(* CoDeSys 2.3.9.41 project: Armen_1.pro *)
(* Libraries: Util.lib 18.5.10 15:14:28, STANDARD.LIB 4.10.05 11:14:46, IECSFC.LIB 13.4.06 15:51:28, SYSLIBTIME.LIB 20.2.06 12:31:16, SYSTASKINFO.LIB 20.2.06 12:31:38, ANALYZATION.LIB 5.10.99 09:05:06, SYSLIBCALLBACK.LIB 20.2.06 12:31:08, PID_Regulators.lib 28.12.06 16:47:54 *)

(* PLC configuration (modules and I/O channels)
Fast discrete inputs [I_SIMPLE_INPUT] node 0, in %IB0 out %QB0 {ChannellName = Fast discrete inputs; Filtrationtime = 10000}
  AT %IX0.0 [BitInput] Discrete input 1 {ChannellName = Enter name}
  AT %IX0.1 [BitInput] Discrete input 2 {ChannellName = Enter name}
AT %IB1.0 [ByteInput] 8 discrete inputs {ChannellName = Enter name}
AT %IB1.1 [ByteInput] 8 discrete inputs {ChannellName = Enter name}
Fan AT %QX2.0 [BitOutput] Fast discrete output 1 {ChannellName = Enter name}
Hot_fan AT %QX2.1 [BitOutput] Fast discrete output 2 {ChannellName = Enter name}
Fan_wall AT %QX2.2 [BitOutput] Fast discrete output 3 {ChannellName = Enter name}
Light_out AT %QX2.3 [BitOutput] Fast discrete output 4 {ChannellName = Enter name}
AT %QB3.0 [ByteOutput] 8 discrete outputs {ChannellName = Enter name}
AT %IX4.0 [BitInput] Special input {ChannellName = Enter name}
AT %QX5.0 [BitOutput] Special output {ChannellName = Enter name}
RS-232 [COM2_USART] node 0, in %IB6.0.0 out %QB6.0.0 {ChannellName = RS-232; CommunicationSpeed = 57600; Parity = NO PARITY CHECK; BitLength = 8 bits; StopLength = One stop bit; InterfaceType = RS232; FrameOriented = RTU; Timeout = 0; Visibility = No}
AT %QB6.1.0 [ByteOutput] {ChannellName = Enter name}
AT %QB6.2.0 [ByteOutput] {ChannellName = Enter name}
AT %QB6.3.0 [ByteOutput] {ChannellName = Enter name}
8 bits [8Bit] node 4, in %IB6.4 out %QB6.4 {ChannellName = 8 bit}
  AT %QB6.4.0 [ByteOutput] {ChannellName = Enter name}
8 bits [8Bit] node 5, in %IB6.5 out %QB6.5 {ChannellName = 8 bit}
  AT %QB6.5.0 [ByteOutput] {ChannellName = Enter name}
8 bits [8Bit] node 6, in %IB6.6 out %QB6.6 {ChannellName = 8 bit}
  AT %QB6.6.0 [ByteOutput] {ChannellName = Enter name}
2 byte [Register] node 7, in %IB6.7 out %QB6.7 {ChannellName = 2 byte}
  Hour_p AT %QW6.7.0 [WordOutput] {ChannellName = Enter name}
2 byte [Register] node 8, in %IB6.8 out %QB6.8 {ChannellName = 2 byte}
  Min_p AT %QW6.8.0 [WordOutput] {ChannellName = Enter name}
2 byte [Register] node 9, in %IB6.9 out %QB6.9 {ChannellName = 2 byte}
  FanWall_t_start AT %QW6.9.0 [WordOutput] {ChannellName = Enter name}
2 byte [Register] node 10, in %IB6.10 out %QB6.10 {ChannellName = 2 byte}
  FanWall_t_stop AT %QW6.10.0 [WordOutput] {ChannellName = Enter name}
2 byte [Register] node 11, in %IB6.11 out %QB6.11 {ChannellName = 2 byte}
  Wind_set AT %QW6.11.0 [WordOutput] {ChannellName = Enter name}
2 byte [Register] node 12, in %IB6.12 out %QB6.12 {ChannellName = 2 byte}
  Wind_Hyst AT %QW6.12.0 [WordOutput] {ChannellName = Enter name}
2 byte [Register] node 13, in %IB6.13 out %QB6.13 {ChannellName = 2 byte}
  Fan_set AT %QW6.13.0 [WordOutput] {ChannellName = Enter name}
2 byte [Register] node 14, in %IB6.14 out %QB6.14 {ChannellName = 2 byte}
  Fan_Hyst AT %QW6.14.0 [WordOutput] {ChannellName = Enter name}
2 byte [Register] node 15, in %IB6.15 out %QB6.15 {ChannellName = 2 byte}
  Hot_set AT %QW6.15.0 [WordOutput] {ChannellName = Enter name}
2 byte [Register] node 16, in %IB6.16 out %QB6.16 {ChannellName = 2 byte}
  Hot_Hyst AT %QW6.16.0 [WordOutput] {ChannellName = Enter name}
2 byte [Register] node 17, in %IB6.17 out %QB6.17 {ChannellName = 2 byte}
  Cold_set AT %QW6.17.0 [WordOutput] {ChannellName = Enter name}
2 byte [Register] node 18, in %IB6.18 out %QB6.18 {ChannellName = 2 byte}
  Cold_hyst AT %QW6.18.0 [WordOutput] {ChannellName = Enter name}
2 byte [Register] node 19, in %IB6.19 out %QB6.19 {ChannellName = 2 byte}
  m_Light_on AT %QW6.19.0 [WordOutput] {ChannellName = Enter name}
2 byte [Register] node 20, in %IB6.20 out %QB6.20 {ChannellName = 2 byte}
  h_light_on AT %QW6.20.0 [WordOutput] {ChannellName = Enter name}
2 byte [Register] node 21, in %IB6.21 out %QB6.21 {ChannellName = 2 byte}
  m_light_off AT %QW6.21.0 [WordOutput] {ChannellName = Enter name}
2 byte [Register] node 22, in %IB6.22 out %QB6.22 {ChannellName = 2 byte}
  h_light_off AT %QW6.22.0 [WordOutput] {ChannellName = Enter name}
2 byte [Register] node 23, in %IB6.23 out %QB6.23 {ChannellName = 2 byte}
  t_tep_i AT %QW6.23.0 [WordOutput] {ChannellName = Enter name}
2 byte [Register] node 24, in %IB6.24 out %QB6.24 {ChannellName = 2 byte}
  v_tep_i AT %QW6.24.0 [WordOutput] {ChannellName = Enter name}
2 byte [Register] node 25, in %IB6.25 out %QB6.25 {ChannellName = 2 byte}
  t_ul_i AT %QW6.25.0 [WordOutput] {ChannellName = Enter name}
2 byte [Register] node 26, in %IB6.26 out %QB6.26 {ChannellName = 2 byte}
  v_ul_i AT %QW6.26.0 [WordOutput] {ChannellName = Enter name}
2 byte [Register] node 27, in %IB6.27 out %QB6.27 {ChannellName = 2 byte}
  AT %QW6.27.0 [WordOutput] {ChannellName = Enter name}
2 byte [Register] node 28, in %IB6.28 out %QB6.28 {ChannellName = 2 byte}
  AT %QW6.28.0 [WordOutput] {ChannellName = Enter name}
2 byte [Register] node 29, in %IB6.29 out %QB6.29 {ChannellName = 2 byte}
  AT %QW6.29.0 [WordOutput] {ChannellName = Enter name}
2 byte [Register] node 30, in %IB6.30 out %QB6.30 {ChannellName = 2 byte}
  AT %QW6.30.0 [WordOutput] {ChannellName = Enter name}
2 byte [Register] node 31, in %IB6.31 out %QB6.31 {ChannellName = 2 byte}
  AT %QW6.31.0 [WordOutput] {ChannellName = Enter name}
4 byte [FourBytes] node 32, in %IB6.32 out %QB6.32 {ChannellName = 4 byte}
  AT %QD6.32.0 [DWordOutput] {ChannellName = Enter name}
AT %QD7.0 [DWordOutput] Last address {ChannellName = Enter name}
AT %QW7.1 [WordOutput] Last error {ChannellName = Enter name}
RS-485-1 [COM1_USART] node 0, in %IB7.0 out %QB7.0 {ChannellName = RS-485-1; CommunicationSpeed = 38400; Parity = NO PARITY CHECK; BitLength = 8 bits; StopLength = One stop bit; InterfaceType = RS485; FrameOriented = ASCII; Timeout = 0; Visibility = No}
Universal Modbus device [ID2000] node 1, in %IB7.1 out %QB7.1 {ChannellName = Universal Modbus device; ModuleIP = 10:0:0:223; ServiceTimeout = 150; TCPport = 502; NetMode = Serial; ModuleSlaveAddress = 2; RequestType = By poll time; PeriodOfService = 100; Visibility = No; RepeatCounter = 0; ByteSequence = Trace_mode}
  AT %QB7.1.0 [ComChannel] Command (0xff - Start) {ChannellName = Enter name}
Wind AT %QD7.1.0.0 [FloatOutput] {ChannellName = Enter name}
AT %QD7.1.1.0 [FloatOutput] {ChannellName = Enter name}
Universal Modbus device [ID2000] node 2, in %IB7.2 out %QB7.2 {ChannellName = Universal Modbus device; ModuleIP = 10:0:0:223; ServiceTimeout = 150; TCPport = 502; NetMode = Serial; ModuleSlaveAddress = 1; RequestType = By poll time; PeriodOfService = 100; Visibility = No; RepeatCounter = 0; ByteSequence = Trace_mode}
  AT %QB7.2.0 [ComChannel] Command (0xff - Start) {ChannellName = Enter name}
t_tep AT %QW7.2.0.0 [WordOutput] {ChannellName = Enter name}
v_tep AT %QW7.2.1.0 [WordOutput] {ChannellName = Enter name}
Universal Modbus device [ID2000] node 3, in %IB7.3 out %QB7.3 {ChannellName = Universal Modbus device; ModuleIP = 10:0:0:223; ServiceTimeout = 150; TCPport = 502; NetMode = Serial; ModuleSlaveAddress = 1; RequestType = By poll time; PeriodOfService = 100; Visibility = No; RepeatCounter = 0; ByteSequence = Trace_mode}
  AT %QB7.3.0 [ComChannel] Command (0xff - Start) {ChannellName = Enter name}
t_ul AT %QW7.3.0.0 [WordOutput] {ChannellName = Enter name}
v_ul AT %QW7.3.1.0 [WordOutput] {ChannellName = Enter name}
AT %QB7.4.0 [ComChannel] Command (0xff - Start) {ChannellName = Enter name}
PR100_in AT %QW7.4.0.0 [WordOutput] {ChannellName = Enter name}
PR100_out AT %QW7.4.1.0 [WordOutput] {ChannellName = Enter name}
Real input module [ID2007] node 2, in %IB7.4.2 out %QB7.4.2 {ChannellName = float input module; ModbusAddress = 0; Command_read_regs = Read holding Registers  (0x03); Visibility = No}
  AT %QD7.4.2.0 [FloatOutput] {ChannellName = Enter name}
Real input module [ID2007] node 3, in %IB7.4.3 out %QB7.4.3 {ChannellName = float input module; ModbusAddress = 0; Command_read_regs = Read holding Registers  (0x03); Visibility = No}
  AT %QD7.4.3.0 [FloatOutput] {ChannellName = Enter name}
*)

(* POU PLC_PRG, CFC *)
PROGRAM PLC_PRG
VAR
	Tof_Cold: TOF;
	FanWall: BLINK;
	Window_contr: HYSTERESIS;
	Hot_contr: HYSTERESIS;
	Cold_contr: HYSTERESIS;
	Tof_hot: TOF;

	Tof_wind: TOF;
	Window2_tim,Window2_tim_2: TON;
END_VAR
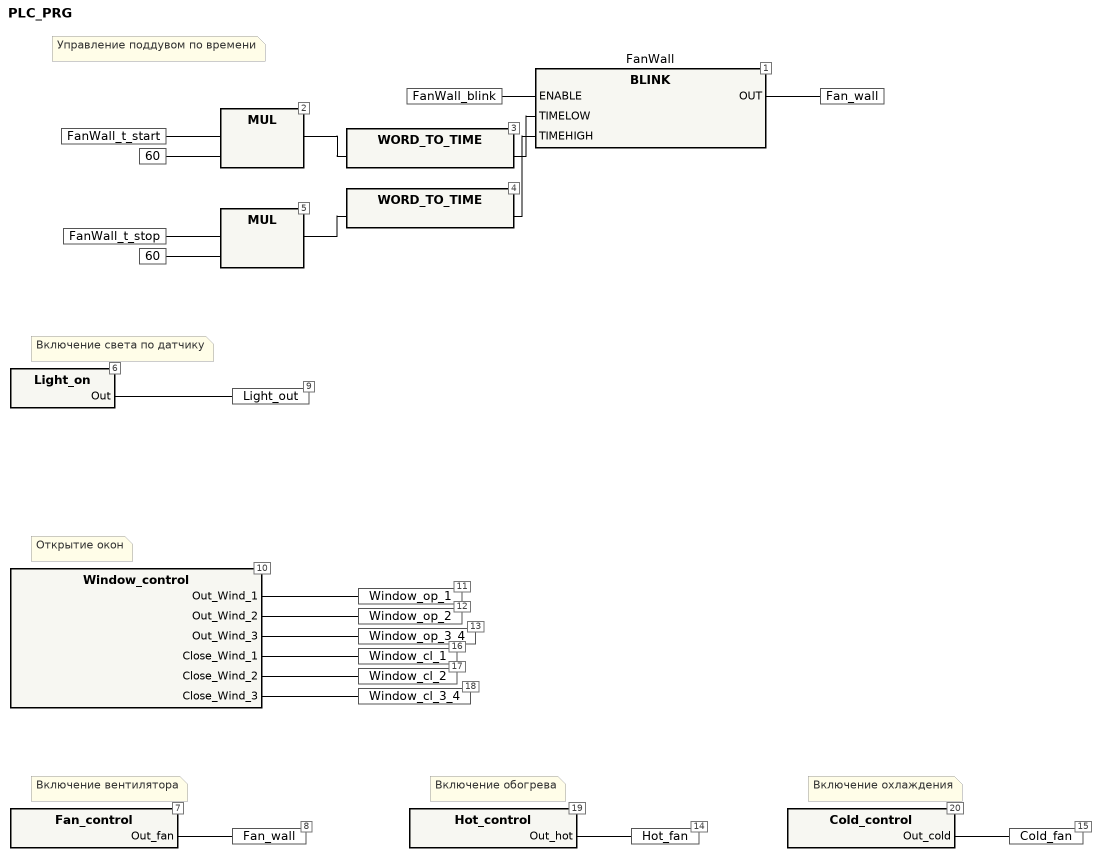
_CFC_ (* Continuous Function Chart, elements in execution order *)
(* Управление поддувом по времени *)
#0 Fan_wall <= #1.OUT
#1 FanWall:BLINK(ENABLE: FanWall_blink, TIMELOW: #3, TIMEHIGH: #4)
#2 MUL(FanWall_t_start, 60)
#3 WORD_TO_TIME(#2)
#4 WORD_TO_TIME(#5)
#5 MUL(FanWall_t_stop, 60)
(* Включение света по датчику *)
#6 Light_on()
#7 Fan_control()
#8 Fan_wall <= #7.Out_fan
#9 Light_out <= #6.Out
#10 Window_control()
#11 Window_op_1 <= #10.Out_Wind_1
#12 Window_op_2 <= #10.Out_Wind_2
#13 Window_op_3_4 <= #10.Out_Wind_3
(* Открытие окон *)
(* Включение вентилятора *)
#14 Hot_fan <= #19.Out_hot
(* Включение обогрева *)
#15 Cold_fan <= #20.Out_cold
(* Включение охлаждения *)
#16 Window_cl_1 <= #10.Close_Wind_1
#17 Window_cl_2 <= #10.Close_Wind_2
#18 Window_cl_3_4 <= #10.Close_Wind_3
#19 Hot_control()
#20 Cold_control()
_END_CFC_
END_PROGRAM

(* POU Light_on, ST *)
PROGRAM Light_on
VAR
END_VAR
VAR_OUTPUT
	Out: BOOL;
END_VAR
IF Light_auto=1 THEN
	IF Light_str_sensor=1 THEN
		Out:=Light_str_sensor;
	END_IF

	IF (Light_str_sensor=0)  THEN
		IF ((m_Light_on+h_Light_on*100)<(Min_p+Hour_p*100)) OR ( (m_Light_off+h_Light_off*100)>(Min_p+Hour_p*100)) THEN
			Out:=1;
		ELSE
			Out:=0;
		END_IF
	END_IF

ELSE
	Light_str_sensor:=0;
	Out:=Light_r;
END_IF
END_PROGRAM

(* POU Fan_control, ST *)
PROGRAM Fan_control
VAR
	Hyst: HYSTERESIS;
	 flag, flag2: BOOL;
	T1: TON;
END_VAR
VAR_OUTPUT
	Out_fan: BOOL;
END_VAR
IF Fan_auto=1 THEN
T1(PT:= T#20s);
Hyst(IN:=REAL_TO_INT(t_tep) *10*(-1));
Hyst.HIGH:= WORD_TO_INT(Fan_set+Fan_Hyst/2)*(-1);
Hyst.low:=WORD_TO_INT( Fan_set-Fan_Hyst/2)*(-1);

	IF flag=0 THEN
		IF Out_fan=1 THEN
			flag:=1;
		END_IF
	ELSE
		IF Out_fan=0 THEN
			flag2:=1;
		END_IF
	END_IF


	IF flag2=1 THEN
		flag:=NOT T1.Q;
		flag2:=NOT T1.Q;
	END_IF

	T1.IN:=flag2;


	Out_fan:=Hyst.OUT AND (NOT flag2);
	Fan_r:=0;
ELSE
	Out_fan:=Fan_r;
END_IF
END_PROGRAM

(* POU Window_control, ST *)
PROGRAM Window_control
VAR
	Hyst: HYSTERESIS;
	 flag, flag2: BOOL;
	T1, Tw_op: TON;
END_VAR
VAR_OUTPUT
	Out_Wind_1, Out_Wind_2, Out_Wind_3: BOOL;
	Close_Wind_1, Close_Wind_2, Close_Wind_3: BOOL;
END_VAR
T1(PT:= T#20s);
Tw_op(PT:= T#20s);
Hyst(IN:=REAL_TO_INT(t_tep) *10*(-1));
Hyst.HIGH:= WORD_TO_INT(Wind_set+Wind_Hyst/2)*(-1);
Hyst.low:=WORD_TO_INT(Wind_set-Wind_Hyst/2)*(-1);

	IF flag=0 THEN
		IF Hyst.OUT=1 THEN
			flag:=1;
		END_IF
	ELSE
		IF Hyst.OUT=0 THEN
			flag2:=1;
		END_IF
	END_IF

	IF wind>50 THEN
		flag2:=1;
	END_IF


	IF flag2=1 THEN
		flag:=NOT T1.Q; (*Сброс таймеров*)
		flag2:=NOT T1.Q;

	END_IF

	T1.IN:=flag2;

	Tw_op.IN:=Hyst.OUT AND (NOT flag2);

	(*Этапы открытия окон*)

	IF Tw_op.PT<t#5s THEN
		Out_Wind_1:=1;
	END_IF


	IF (Tw_op.PT<t#5s) AND (Tw_op.PT<t#10s) THEN
		Out_Wind_2:=1;
		Out_Wind_1:=0;
	END_IF

	IF (Tw_op.PT<t#10s) AND (Tw_op.PT<t#15s) THEN
		Out_Wind_3:=1;
		Out_Wind_2:=0;
	END_IF

	IF ((Hyst.OUT AND (NOT flag2))=FALSE) OR (Tw_op.PT>t#15s) THEN
		Out_Wind_1:=0;
		Out_Wind_2:=0;
		Out_Wind_3:=0;
	END_IF

(*Этапы закрытия окон*)

	IF T1.PT<t#5s THEN
		Close_Wind_1:=1;
	END_IF

	IF (T1.PT<t#5s) AND (T1.PT<t#10s) THEN
		Close_Wind_2:=1;
		Close_Wind_1:=0;
	END_IF

	IF (T1.PT<t#10s) AND (T1.PT<t#15s) THEN
		Close_Wind_3:=1;
		Close_Wind_2:=0;
	END_IF

	IF (Hyst.OUT =TRUE) OR (T1.PT>t#15s) THEN
		Close_Wind_1:=0;
		Close_Wind_2:=0;
		Close_Wind_3:=0;
	END_IF

	IF (Out_Wind_1=1) OR (Out_Wind_2=1) OR ( Out_Wind_3=1) THEN
		Close_Wind_1:=0;
		Close_Wind_2:=0;
		Close_Wind_3:=0;
	END_IF
END_PROGRAM

(* POU Hot_control, ST *)
PROGRAM Hot_control
VAR
	Hyst: HYSTERESIS;
	 flag, flag2: BOOL;
	T1: TON;
END_VAR
VAR_OUTPUT
	Out_hot: BOOL;
END_VAR
IF Hot_auto=1 THEN
T1(PT:= T#20s);
Hyst(IN:=REAL_TO_INT(t_tep) *10);
Hyst.HIGH:= Hot_set+Hot_Hyst/2;
Hyst.low:= Hot_set-Hot_Hyst/2;

	IF flag=0 THEN
		IF Out_hot=1 THEN
			flag:=1;
		END_IF
	ELSE
		IF Out_hot=0 THEN
			flag2:=1;
		END_IF
	END_IF


	IF flag2=1 THEN
		flag:=NOT T1.Q;
		flag2:=NOT T1.Q;
	END_IF

	T1.IN:=flag2;


	Out_hot:=Hyst.OUT AND (NOT flag2);
	Hot_r:=0;
ELSE
	Out_hot:=Hot_r;
END_IF
END_PROGRAM

(* POU Cold_control, ST *)
PROGRAM Cold_control
VAR
	Hyst: HYSTERESIS;
	 flag, flag2: BOOL;
	T1: TON;
END_VAR
VAR_OUTPUT
	Out_cold: BOOL;
END_VAR
IF Cold_auto=1 THEN
T1(PT:= T#20s);
Hyst(IN:=REAL_TO_INT(t_tep) *10*(-1));
Hyst.HIGH:= WORD_TO_INT(Cold_set+Cold_hyst/2)*(-1);
Hyst.low:= WORD_TO_INT(Cold_set-Cold_hyst/2)*(-1);

	IF flag=0 THEN
		IF Out_cold=1 THEN
			flag:=1;
		END_IF
	ELSE
		IF Out_cold=0 THEN
			flag2:=1;
		END_IF
	END_IF


	IF flag2=1 THEN
		flag:=NOT T1.Q;
		flag2:=NOT T1.Q;
	END_IF

	T1.IN:=flag2;


	Out_cold:=Hyst.OUT AND (NOT flag2);
	Cold_r:=0;
ELSE
	Out_cold:=Cold_r;
END_IF
END_PROGRAM

(* POU Mixer, ST *)
PROGRAM Mixer
VAR
	flag: BOOL;
END_VAR
VAR_OUTPUT

END_VAR
	IF Auto_water=0 THEN
		PR100_out.2:=Valv1;
		PR100_out.3:=Valv2;
		PR100_out.4:=Valv3;
		PR100_out.5:=Valv4;
		PR100_out.6:=Valv5;
		PR100_out.7:=Valv6;
		flag:=0;
	ELSE
		IF flag=0 THEN  (*Обнуление выходных сигналов *)
			PR100_out.2:=0;
			PR100_out.3:=0;
			PR100_out.4:=0;
			PR100_out.5:=0;
			PR100_out.6:=0;
			PR100_out.7:=0;
			flag:=1;
		END_IF
	END_IF
END_PROGRAM
